(* CODESYS project TvillingRobotProgram.ecp

Project tree, tasks and I/O mapping:
  Controller : 750-8214 PFC200 G2 2ETH RS CAN, WAGO, order no. 0750-8214, version 5.17.3.10
    application Application
      libraries: ; WagoSysPlainMem, 1.5.2.0 (WAGO); WagoAppCloud, * (WAGO); VisuDialogs, * (System)
      task PLC_Task (cyclic, interval t#50ms, priority 15) calls MQTT_Modbus
      task VISU_TASK (cyclic, interval 100 ms, priority 15) calls VisuElems.Visu_Prg
      program MQTT_Modbus [LD]
      FunctionBlocks/
        function block MQTT_Sub [ST]
        function block MQTT_Pub [ST]
        function block MQTT_To_Modbus [ST]
        function block Modbus_To_MQTT [ST]
        function block Filter_Til_MQTT [ST]
      visualisation TvillingTest
      global variables GVL
      program Modbus_MQTT [LD]
    Kbus : Kbus, WAGO, version 1.4.0.2
        unmapped channels: K-BUS diagnostics
    MODBUS
      MODBUS : MODBUS, WAGO, order no. n/a, version 1.1.1.16
        LocalDeviceModbus : MODBUS Slave, WAGO, order no. n/a, version 1.1.1.16
            settings: OffsetMap = 0; OffsetMap = 32; OffsetMap = 16; OffsetMap = 48; OffsetMap = 64; OffsetMap = 80; OffsetMap = 2080; OffsetMap = 2112; OffsetMap = 2096; OffsetMap = 2128; OffsetMap = 2144; OffsetMap = 2160
            input  Application.GVL.Modbus_Recive_Base : WORD  // 
            input  Application.GVL.Modbus_Recive_Elbow : WORD  // 
            input  Application.GVL.Modbus_Recive_Sholder : WORD  // 
            input  Application.GVL.Modbus_Recive_Wrist1 : WORD  // 
            input  Application.GVL.Modbus_Recive_Wrist2 : WORD  // 
            input  Application.GVL.Modbus_Recive_wrist3 : WORD  // 
            output Application.GVL.Modbus_Send_Base : WORD  // 
            output Application.GVL.Modbus_Send_Elbow : WORD  // 
            output Application.GVL.Modbus_Send_Sholder : WORD  // 
            output Application.GVL.Modbus_Send_Wrist1 : WORD  // 
            output Application.GVL.Modbus_Send_Wrist2 : WORD  // 
            output Application.GVL.Modbus_Send_Wrist3 : WORD  // 
          TcpSettings : Modbus TCP Slave, WAGO, order no. n/a, version 1.1.1.16
              settings: TCP connection watchdog = 200 10ms
    CANbus
    Common.PCI
    EtherNet/IP
      Ethernet : Ethernet, WAGO, version 35.17.0.0
    Serial
      COM1 : COM1, WAGO, version 0.0.0.19
  Generic_Modbus_Master : ThirdParty Modbus Master, WAGO, order no. GenericModbusMaster, version 1.0.0.1
  libraries: Util, * (System)
  text list GlobalTextList
*)

// Controller/Application/GVL
{attribute 'qualified_only'}
VAR_GLOBAL
	Trigger : BOOL;
	// Variabler for å subscribe til MQTT
	MQTT_SubTopic1 : STRING(255) := 'triplet/fromArduino/base';
	MQTT_SubTopic2 : STRING(255) := 'triplet/fromArduino/shoulder';
	MQTT_SubTopic3 : STRING(255) := 'triplet/fromArduino/elbow';
	MQTT_SubTopic4 : STRING(255) := 'triplet/fromArduino/wrist1';
	MQTT_SubTopic5 : STRING(255) := 'triplet/fromArduino/wrist2';
	MQTT_SubTopic6 : STRING(255) := 'triplet/fromArduino/wrist3';
	
	MQTT_V_Base : INT;
	MQTT_V_Shoulder : INT;
	MQTT_V_Elbow : INT;
	MQTT_V_Wrist1 : INT;
	MQTT_V_Wrist2 : INT;
	MQTT_V_Wrist3 : INT;
	
	// Variabler for å publisere til MQTT "Tvilling"
	MQTT_Sim_Topic1 : STRING(255) := 'triplet/simulator/base';
	MQTT_Sim_Topic2 : STRING(255) := 'triplet/simulator/shoulder';
	MQTT_Sim_Topic3 : STRING(255) := 'triplet/simulator/elbow';
	MQTT_Sim_Topic4 : STRING(255) := 'triplet/simulator/wrist1';
	MQTT_Sim_Topic5 : STRING(255) := 'triplet/simulator/wrist2';
	MQTT_Sim_Topic6 : STRING(255) := 'triplet/simulator/wrist3';
	
	// Variabler for å publishe til MQTT
	MQTT_PubTopic1 : STRING(255) := 'triplet/controller/base';
	MQTT_PubTopic2 : STRING(255) := 'triplet/controller/shoulder';
	MQTT_PubTopic3 : STRING(255) := 'triplet/controller/elbow';
	MQTT_PubTopic4 : STRING(255) := 'triplet/controller/wrist1';
	MQTT_PubTopic5 : STRING(255) := 'triplet/controller/wrist2';
	MQTT_PubTopic6 : STRING(255) := 'triplet/controller/wrist3';

	// Variabler til UR10 (Modbus)
	Modbus_Send_Base : WORD;
	Modbus_Send_Sholder : WORD;
	Modbus_Send_Elbow : WORD;
	Modbus_Send_Wrist1 : WORD;
	Modbus_Send_Wrist2 : WORD;
	Modbus_Send_Wrist3 : WORD;
	
	// Variabler fra UR10 (Modbus)
	Modbus_Recive_Base : WORD;
	Modbus_Recive_Sholder : WORD;
	Modbus_Recive_Elbow : WORD;
	Modbus_Recive_Wrist1 : WORD;
	Modbus_Recive_Wrist2 : WORD;
	Modbus_Recive_wrist3 : WORD;
	
	// UR10 Joints
	UR_Base : INT;
	UR_Shoulder : INT;
	UR_Elbow : INT;
	UR_Wrist1 : INT;
	UR_Wrist2 : INT;
	UR_Wrist3 : INT;
END_VAR

// Controller/Application/MQTT_Modbus
PROGRAM MQTT_Modbus
VAR
	MQTT_Max : REAL := 360;
	MQTT_Min : REAL := -360;
	Modbus_Max : REAL := 12660;
	Modbus_Min : REAL := 0;
	Offset : REAL :=360;
	MQTT_PUB_Max : REAL := 360;
	MQTT_PUB_Min : REAL := -360;
	MQTT_Sub_0: MQTT_Sub;
	MQTT_Sub_1: MQTT_Sub;
	MQTT_Sub_2: MQTT_Sub;
	MQTT_Sub_3: MQTT_Sub;
	MQTT_Sub_4: MQTT_Sub;
	MQTT_Sub_5: MQTT_Sub;
	MQTT_To_Modbus_0: MQTT_To_Modbus;
	MQTT_To_Modbus_1: MQTT_To_Modbus;
	MQTT_To_Modbus_2: MQTT_To_Modbus;
	MQTT_To_Modbus_3: MQTT_To_Modbus;
	MQTT_To_Modbus_4: MQTT_To_Modbus;
	MQTT_To_Modbus_5: MQTT_To_Modbus;
	MQTT_To_Modbus_6: MQTT_To_Modbus;
	MQTT_Pub_0: MQTT_Pub;
	MQTT_Pub_1: MQTT_Pub;
	MQTT_Pub_2: MQTT_Pub;
	MQTT_Pub_3: MQTT_Pub;
	MQTT_Pub_4: MQTT_Pub;
	MQTT_Pub_5: MQTT_Pub;
	BLINK_0: BLINK;
	Publish : BOOL;
	BLINK_1: BLINK;
	Filter_Til_MQTT_0: Filter_Til_MQTT;
	Filter_Til_MQTT_1: Filter_Til_MQTT;
	Filter_Til_MQTT_2: Filter_Til_MQTT;
	Filter_Til_MQTT_3: Filter_Til_MQTT;
	Filter_Til_MQTT_4: Filter_Til_MQTT;
	Filter_Til_MQTT_5: Filter_Til_MQTT;
	Update_Value : REAL := 1;
	TOF_0: TOF;
	TOF_1: TOF;
	TOF_2: TOF;
	TOF_3: TOF;
	TOF_4: TOF;
	TOF_5: TOF;
END_VAR

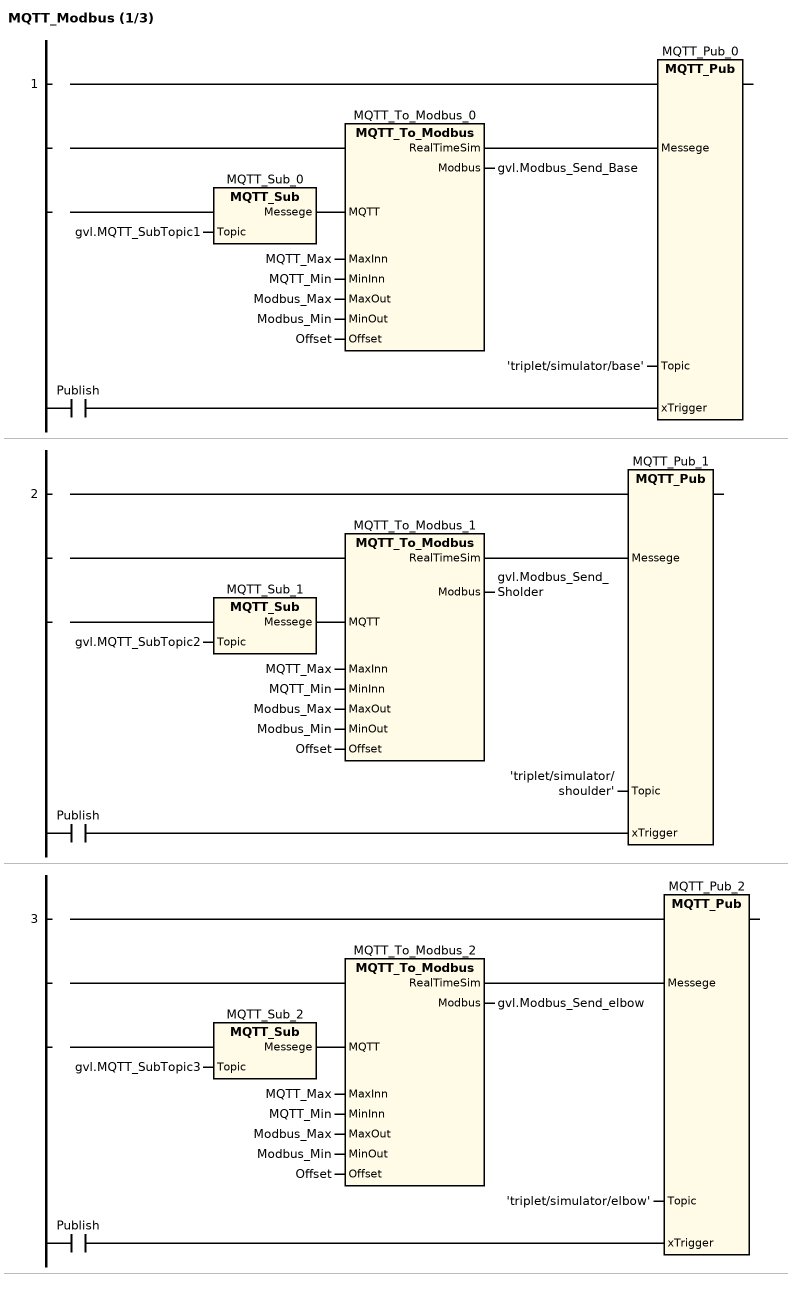
// NETWORK 1
MQTT_Sub_0(Topic := gvl.MQTT_SubTopic1); // MQTT_Sub
MQTT_To_Modbus_0(
    MQTT := MQTT_Sub_0.Messege,
    MaxInn := MQTT_Max,
    MinInn := MQTT_Min,
    MaxOut := Modbus_Max,
    MinOut := Modbus_Min,
    Offset := Offset,
    Modbus => gvl.Modbus_Send_Base); // MQTT_To_Modbus
MQTT_Pub_0(Messege := MQTT_To_Modbus_0.RealTimeSim, Topic := 'triplet/simulator/base', xTrigger := Publish); // MQTT_Pub

// NETWORK 2
MQTT_Sub_1(Topic := gvl.MQTT_SubTopic2); // MQTT_Sub
MQTT_To_Modbus_1(
    MQTT := MQTT_Sub_1.Messege,
    MaxInn := MQTT_Max,
    MinInn := MQTT_Min,
    MaxOut := Modbus_Max,
    MinOut := Modbus_Min,
    Offset := Offset,
    Modbus => gvl.Modbus_Send_Sholder); // MQTT_To_Modbus
MQTT_Pub_1(
    Messege := MQTT_To_Modbus_1.RealTimeSim,
    Topic := 'triplet/simulator/shoulder',
    xTrigger := Publish); // MQTT_Pub

// NETWORK 3
MQTT_Sub_2(Topic := gvl.MQTT_SubTopic3); // MQTT_Sub
MQTT_To_Modbus_2(
    MQTT := MQTT_Sub_2.Messege,
    MaxInn := MQTT_Max,
    MinInn := MQTT_Min,
    MaxOut := Modbus_Max,
    MinOut := Modbus_Min,
    Offset := Offset,
    Modbus => gvl.Modbus_Send_elbow); // MQTT_To_Modbus
MQTT_Pub_2(Messege := MQTT_To_Modbus_2.RealTimeSim, Topic := 'triplet/simulator/elbow', xTrigger := Publish); // MQTT_Pub

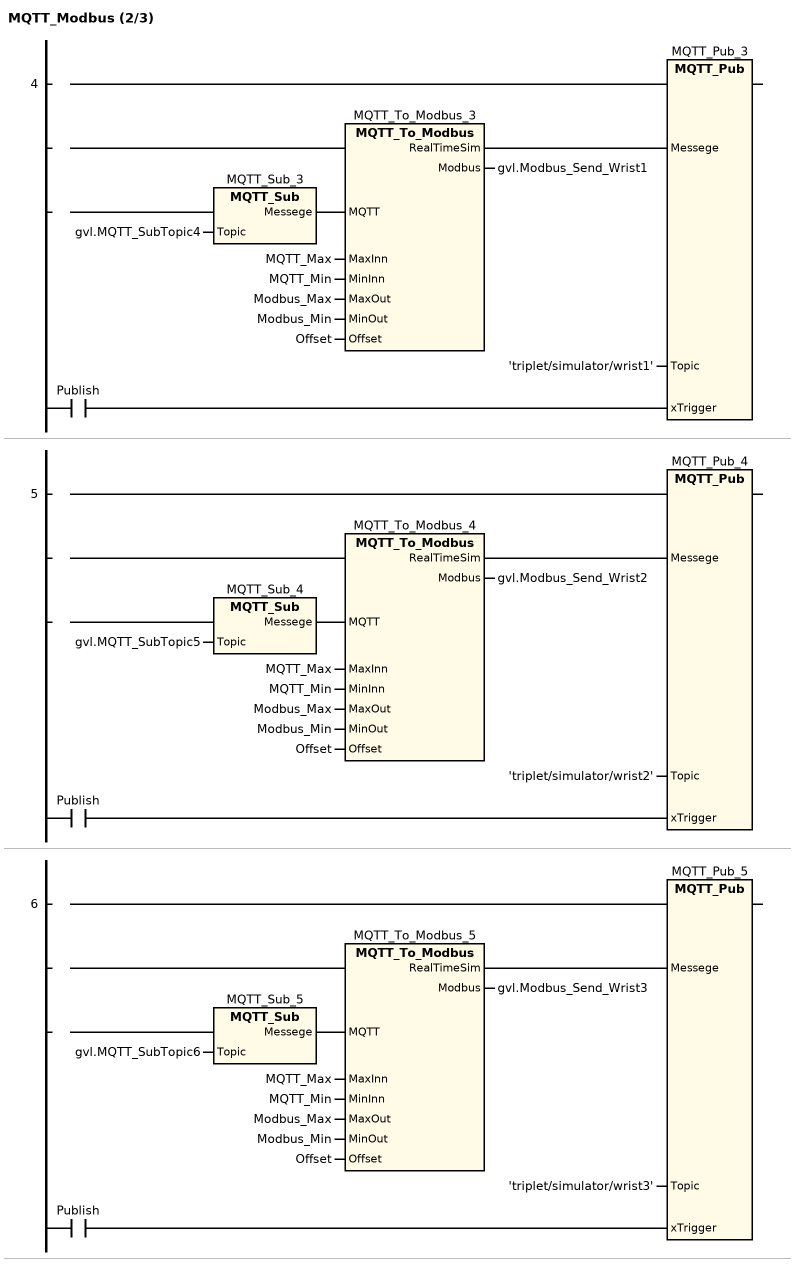
// NETWORK 4
MQTT_Sub_3(Topic := gvl.MQTT_SubTopic4); // MQTT_Sub
MQTT_To_Modbus_3(
    MQTT := MQTT_Sub_3.Messege,
    MaxInn := MQTT_Max,
    MinInn := MQTT_Min,
    MaxOut := Modbus_Max,
    MinOut := Modbus_Min,
    Offset := Offset,
    Modbus => gvl.Modbus_Send_Wrist1); // MQTT_To_Modbus
MQTT_Pub_3(Messege := MQTT_To_Modbus_3.RealTimeSim, Topic := 'triplet/simulator/wrist1', xTrigger := Publish); // MQTT_Pub

// NETWORK 5
MQTT_Sub_4(Topic := gvl.MQTT_SubTopic5); // MQTT_Sub
MQTT_To_Modbus_4(
    MQTT := MQTT_Sub_4.Messege,
    MaxInn := MQTT_Max,
    MinInn := MQTT_Min,
    MaxOut := Modbus_Max,
    MinOut := Modbus_Min,
    Offset := Offset,
    Modbus => gvl.Modbus_Send_Wrist2); // MQTT_To_Modbus
MQTT_Pub_4(Messege := MQTT_To_Modbus_4.RealTimeSim, Topic := 'triplet/simulator/wrist2', xTrigger := Publish); // MQTT_Pub

// NETWORK 6
MQTT_Sub_5(Topic := gvl.MQTT_SubTopic6); // MQTT_Sub
MQTT_To_Modbus_5(
    MQTT := MQTT_Sub_5.Messege,
    MaxInn := MQTT_Max,
    MinInn := MQTT_Min,
    MaxOut := Modbus_Max,
    MinOut := Modbus_Min,
    Offset := Offset,
    Modbus => gvl.Modbus_Send_Wrist3); // MQTT_To_Modbus
MQTT_Pub_5(Messege := MQTT_To_Modbus_5.RealTimeSim, Topic := 'triplet/simulator/wrist3', xTrigger := Publish); // MQTT_Pub

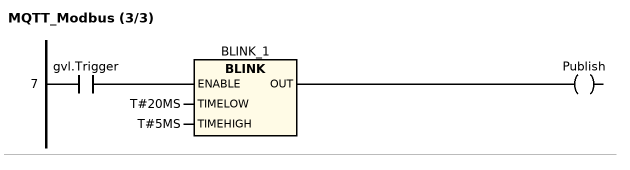
// NETWORK 7
BLINK_1(ENABLE := gvl.Trigger, TIMELOW := T#20MS, TIMEHIGH := T#5MS); // BLINK
Publish := BLINK_1.OUT;

END_PROGRAM

// Controller/Application/FunctionBlocks/MQTT_Pub
FUNCTION_BLOCK MQTT_Pub
VAR_INPUT
	Messege : STRING;
	Topic : STRING(255);
	xTrigger : BOOL;
END_VAR
VAR_OUTPUT
END_VAR
VAR
	sPub:STRING:='TESTSjur';
	FB_Pub : WagoAppCloud.FbPublishMQTT;
	aData: ARRAY [0..100] OF BYTE; 
	xError_Pub: BOOL;
END_VAR

wagoSysPlainMem.MemCopy( pDest:= ADR (aData), pSource:=ADR(Messege), udiSize:=LEN(Messege) );



FB_Pub(
    sTopic:=Topic , 
    eQualityOfService:= , 
    xRetain:= , 
    dwSize:= LEN(Messege), 
    aData:=aData , 
    xTrigger:= xTrigger, 
    xBusy=> , 
    xError=> xError_Pub , 
    oStatus=> );

END_FUNCTION_BLOCK

// Controller/Application/FunctionBlocks/MQTT_To_Modbus
FUNCTION_BLOCK MQTT_To_Modbus
VAR_INPUT
	MQTT : INT;
	MaxInn : REAL;
	MinInn : REAL;
	MaxOut : REAL;
	MinOut : REAL;
	Offset : REAL;
END_VAR
VAR_OUTPUT
	RealTimeSim : STRING;
	Modbus : WORD;
END_VAR
VAR
	Sim_L : REAL;
	MQTT_L : REAL;
	Modbus_L : REAL;
END_VAR

MQTT_L := INT_TO_REAL(MQTT);

Modbus_L := ((MQTT_L+offset)*((MaxOut-MinOut)/((MaxInn+offset)-(MinInn+offset))));

RealTimeSim := REAL_TO_STRING(MQTT_L);
Modbus := REAL_TO_WORD(Modbus_L);

END_FUNCTION_BLOCK

// Controller/Application/FunctionBlocks/MQTT_Sub
FUNCTION_BLOCK MQTT_Sub
VAR_INPUT
	Topic : STRING(255);
END_VAR
VAR_OUTPUT
	Messege: INT;
END_VAR
VAR
	FB_Sub:WagoAppCloud.FbSubscribeMQTT;
    xSubscribe: BOOL:=TRUE; 

    aPayloadData: ARRAY [0..100] OF BYTE; 
    xError_Sub: BOOL;
    xDataReceived :BOOL;
    dwReceivedBytes:DWORD;
    sSub:STRING(255);
END_VAR

FB_Sub(
    xSubscribe:=xSubscribe , 
    sTopic:=Topic , 
    eQoS:= , 
    aPayloadData:= aPayloadData, 
    xBusy=> , 
    xError=> xError_Sub, 
    oStatus=> , 
    xDataReceived=>xDataReceived , 
    dwRxNBytes=>dwReceivedBytes, 
    xDataTruncated=> , 
    sReceivedTopic=> );
    wagoSysPlainMem.MemCopySecure(pDest:=ADR(sSub), udiDestSize:=255 ,pSource:=ADR(aPayloadData),udiSourceSize:=dwReceivedBytes,bPadding:=0);
	
	Messege := STRING_TO_INT(sSub);

END_FUNCTION_BLOCK

// Controller/Application/FunctionBlocks/Filter_Til_MQTT
FUNCTION_BLOCK Filter_Til_MQTT
VAR_INPUT
	input : REAL;
	Update_Value : REAL;
END_VAR
VAR_OUTPUT
	Output : STRING;
	Update : BOOL;
END_VAR
VAR
	Old_Value : REAL;
END_VAR

IF input < (Old_Value + Update_Value)
	THEN
	Output := REAL_TO_STRING(input);
	Old_Value := input;
	Update := TRUE;
	ELSIF input > (Old_Value - Update_Value)
		THEN
		Output := REAL_TO_STRING(input);
		Old_Value := input;
		Update := TRUE;
		END_IF
		
Update := FALSE;

END_FUNCTION_BLOCK

// Controller/Application/Modbus_MQTT
PROGRAM Modbus_MQTT
VAR
	Publish : BOOL;
	MQTT_Max : REAL := 720;
	MQTT_Min : REAL := 0;
	Modbus_Max : REAL := 12660;
	Modbus_Min : REAL := 0;
	UR_Max : REAL := 720;
	UR_Min : REAL := 0;
	MQTT_Pub_0: MQTT_Pub;
	MQTT_Pub_1: MQTT_Pub;
	MQTT_Pub_2: MQTT_Pub;
	MQTT_Pub_3: MQTT_Pub;
	MQTT_Pub_4: MQTT_Pub;
	MQTT_Pub_5: MQTT_Pub;
	Modbus_To_MQTT_0: Modbus_To_MQTT;
	Modbus_To_MQTT_1: Modbus_To_MQTT;
	Modbus_To_MQTT_2: Modbus_To_MQTT;
	Modbus_To_MQTT_3: Modbus_To_MQTT;
	Modbus_To_MQTT_4: Modbus_To_MQTT;
	Modbus_To_MQTT_5: Modbus_To_MQTT;
	BLINK_0: BLINK;
END_VAR

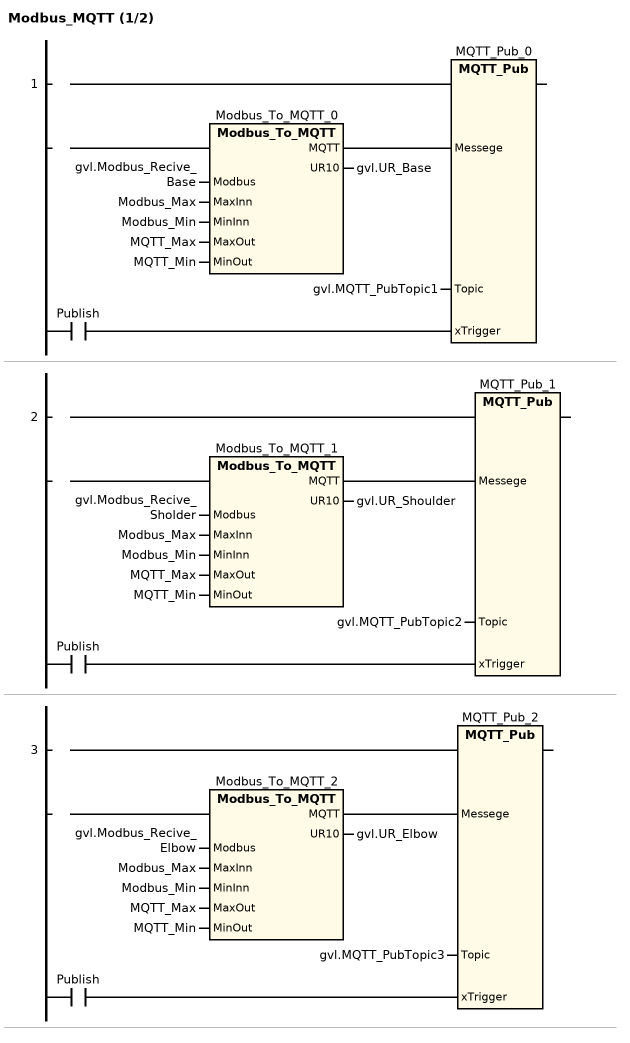
// NETWORK 1
Modbus_To_MQTT_0(
    Modbus := gvl.Modbus_Recive_Base,
    MaxInn := Modbus_Max,
    MinInn := Modbus_Min,
    MaxOut := MQTT_Max,
    MinOut := MQTT_Min,
    UR10 => gvl.UR_Base); // Modbus_To_MQTT
MQTT_Pub_0(Messege := Modbus_To_MQTT_0.MQTT, Topic := gvl.MQTT_PubTopic1, xTrigger := Publish); // MQTT_Pub

// NETWORK 2
Modbus_To_MQTT_1(
    Modbus := gvl.Modbus_Recive_Sholder,
    MaxInn := Modbus_Max,
    MinInn := Modbus_Min,
    MaxOut := MQTT_Max,
    MinOut := MQTT_Min,
    UR10 => gvl.UR_Shoulder); // Modbus_To_MQTT
MQTT_Pub_1(Messege := Modbus_To_MQTT_1.MQTT, Topic := gvl.MQTT_PubTopic2, xTrigger := Publish); // MQTT_Pub

// NETWORK 3
Modbus_To_MQTT_2(
    Modbus := gvl.Modbus_Recive_Elbow,
    MaxInn := Modbus_Max,
    MinInn := Modbus_Min,
    MaxOut := MQTT_Max,
    MinOut := MQTT_Min,
    UR10 => gvl.UR_Elbow); // Modbus_To_MQTT
MQTT_Pub_2(Messege := Modbus_To_MQTT_2.MQTT, Topic := gvl.MQTT_PubTopic3, xTrigger := Publish); // MQTT_Pub

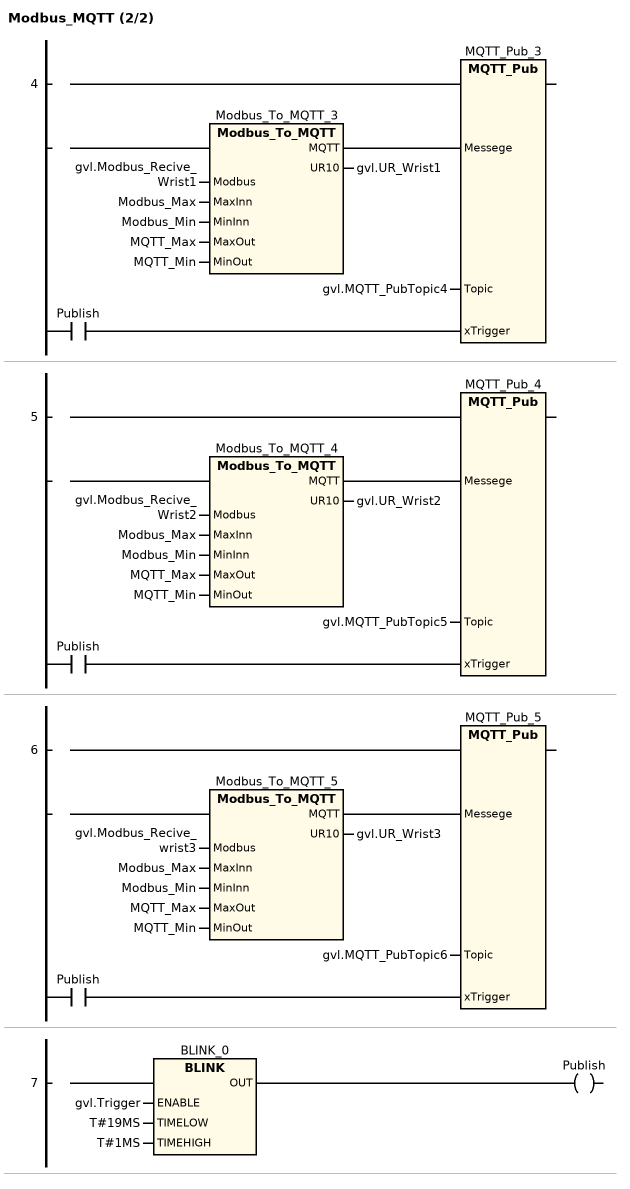
// NETWORK 4
Modbus_To_MQTT_3(
    Modbus := gvl.Modbus_Recive_Wrist1,
    MaxInn := Modbus_Max,
    MinInn := Modbus_Min,
    MaxOut := MQTT_Max,
    MinOut := MQTT_Min,
    UR10 => gvl.UR_Wrist1); // Modbus_To_MQTT
MQTT_Pub_3(Messege := Modbus_To_MQTT_3.MQTT, Topic := gvl.MQTT_PubTopic4, xTrigger := Publish); // MQTT_Pub

// NETWORK 5
Modbus_To_MQTT_4(
    Modbus := gvl.Modbus_Recive_Wrist2,
    MaxInn := Modbus_Max,
    MinInn := Modbus_Min,
    MaxOut := MQTT_Max,
    MinOut := MQTT_Min,
    UR10 => gvl.UR_Wrist2); // Modbus_To_MQTT
MQTT_Pub_4(Messege := Modbus_To_MQTT_4.MQTT, Topic := gvl.MQTT_PubTopic5, xTrigger := Publish); // MQTT_Pub

// NETWORK 6
Modbus_To_MQTT_5(
    Modbus := gvl.Modbus_Recive_wrist3,
    MaxInn := Modbus_Max,
    MinInn := Modbus_Min,
    MaxOut := MQTT_Max,
    MinOut := MQTT_Min,
    UR10 => gvl.UR_Wrist3); // Modbus_To_MQTT
MQTT_Pub_5(Messege := Modbus_To_MQTT_5.MQTT, Topic := gvl.MQTT_PubTopic6, xTrigger := Publish); // MQTT_Pub

// NETWORK 7
BLINK_0(ENABLE := gvl.Trigger, TIMELOW := T#19MS, TIMEHIGH := T#1MS); // BLINK
Publish := BLINK_0.OUT;

END_PROGRAM

// Controller/Application/FunctionBlocks/Modbus_To_MQTT
FUNCTION_BLOCK Modbus_To_MQTT
VAR_INPUT
	Modbus : WORD;
	MaxInn : REAL;
	MinInn : REAL;
	MaxOut : REAL;
	MinOut : REAL;
END_VAR
VAR_OUTPUT
	MQTT : STRING;
	UR10 : INT;
END_VAR
VAR
	MQTT_L : REAL;
	Modbus_L : REAL;
	UR10_L : REAL;
END_VAR

Modbus_L := WORD_TO_REAL(Modbus);

MQTT_L := (Modbus_L*((MaxOut-MinOut)/(MaxInn-MinInn)));
UR10_L := (Modbus_L * ((MaxOut - MinOut)/(MaxInn - MinInn)));


MQTT := REAL_TO_STRING(MQTT_L-360);
UR10 := REAL_TO_INT(UR10_L-360);

END_FUNCTION_BLOCK

// Controller/Application/TvillingTest
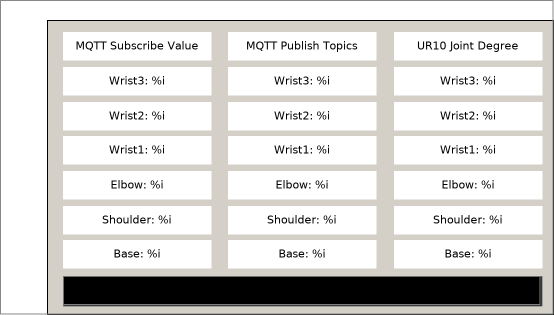
VISUALIZATION TvillingTest  // 554x315
    Rectangle (47,20 507x295)
    Textfield (62,31 150x30), "MQTT Subscribe Value"
    Textfield (62,66 150x30), "Wrist3: %i", text variable: GVL.MQTT_V_Wrist3
        OnMouseClick: write the text variable via VisuDialogs.Keypad
    Textfield (62,101 150x30), "Wrist2: %i", text variable: GVL.MQTT_V_Wrist2
        OnMouseClick: write the text variable via VisuDialogs.Keypad
    Textfield (62,135 150x30), "Wrist1: %i", text variable: GVL.MQTT_V_Wrist1
        OnMouseClick: write the text variable via VisuDialogs.Keypad
    Textfield (62,170 150x30), "Elbow: %i", text variable: GVL.MQTT_V_Elbow
        OnMouseClick: write the text variable via VisuDialogs.Keypad
    Textfield (62,205 150x30), "Shoulder: %i", text variable: GVL.MQTT_V_Shoulder
        OnMouseClick: write the text variable via VisuDialogs.Keypad
    Textfield (62,239 150x30), "Base: %i", text variable: GVL.MQTT_V_Base
        OnMouseClick: write the text variable via VisuDialogs.Keypad
    Textfield (227,31 150x30), "MQTT Publish Topics"
    Textfield (227,66 150x30), "Wrist3: %i", text variable: GVL.MQTT_Sim_Topic6
        OnMouseClick: write the text variable via VisuDialogs.Keypad
    Textfield (227,101 150x30), "Wrist2: %i", text variable: GVL.MQTT_Sim_Topic5
        OnMouseClick: write the text variable via VisuDialogs.Keypad
    Textfield (227,135 150x30), "Wrist1: %i", text variable: GVL.MQTT_Sim_Topic4
        OnMouseClick: write the text variable via VisuDialogs.Keypad
    Textfield (227,170 150x30), "Elbow: %i", text variable: GVL.MQTT_Sim_Topic3
        OnMouseClick: write the text variable via VisuDialogs.Keypad
    Textfield (227,205 150x30), "Shoulder: %i", text variable: GVL.MQTT_Sim_Topic2
        OnMouseClick: write the text variable via VisuDialogs.Keypad
    Textfield (227,239 150x30), "Base: %i", text variable: GVL.MQTT_Sim_Topic1
        OnMouseClick: write the text variable via VisuDialogs.Keypad
    Textfield (393,31 150x30), "UR10 Joint Degree"
    Textfield (393,66 150x30), "Wrist3: %i", text variable: GVL.UR_Wrist3
    Textfield (393,101 150x30), "Wrist2: %i", text variable: GVL.UR_Wrist2
    Textfield (393,135 150x30), "Wrist1: %i", text variable: GVL.UR_Wrist1
    Textfield (393,170 150x30), "Elbow: %i", text variable: GVL.UR_Elbow
    Textfield (393,205 150x30), "Shoulder: %i", text variable: GVL.UR_Shoulder
    Textfield (393,239 150x30), "Base: %i", text variable: GVL.UR_Base
    Button (63,276 479x30), "Enable Publishing to MQTT"
        toggle GVL.Trigger
END_VISUALIZATION
